INTERFACE I_XTS

METHOD RegisterMovers : HRESULT
VAR_INPUT
	MyMover : ITF_XtsMoverAxis;
END_VAR
END_METHOD

END_INTERFACE

(* stored: Version 1.1.0.1
   Itf I_XTS: Id {eb22a7d8-6cc9-41fe-bacb-ecb9c288212d}
   Method RegisterMovers: Id {e65bc655-b1b5-4ed3-91eb-2d51871a4d75} *)
